//{attribute 'qualified_only'}
{attribute 'strict'}
TYPE E_InverterStatusWord :
(
	eSLF1      := 568,	// błąd komunikacja Modbus przerwana i nieaktywna
	enSL	   := 592,	// Stan po udanym resecie błędu komunikacji komedną eResetInv = 128
	eRdy       := 561,	// Stan po ustawieniu gotowości Inverta komendą eReady = 14
	eZeroSpeed := 567,  // Stan po ustawieniu komendy eFwd = 15 lub eRev = 2063 gdy jest zerowa prędkośc zadana speed = 0 
	eFwdOper   := 1591, // Stan gdy napęd pracuje w kierunku przodu po komendzie eFwd = 15 i osiągnał zadaną prędkość
	eRevOper   := 34359	// Stan gdy napęd pracuje w kierunku odwrotnym po komendzie eRev = 2063 i osiągnał zadaną prędkość 	
	
)WORD;
END_TYPE

(* stored: Version 1.1.0.1, ProductVersion 3.1.4024.12
   EnumerationTextList E_InverterStatusWord: Id {a537bab2-a1fa-4c2f-8f0c-222f1e9a65c9} *)
